ABB RobotStudio station: TEST1_20190225-105659.rsstn

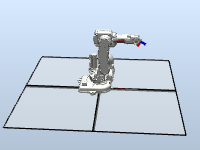
Station TEST1 (saved by RobotStudio 6.8.8148.134)
Controller IRB_140_6kg_0.81m
  mechanical unit ROB_1: IRB140_6_81_C_03, 6 joints, base frame (0, 0, 0) mm
Layout (positions relative to the parent item):
  - IRB140_6_81_C_03 [mechanism, from Robots\IRB140_6_81_C_G_03.rslib] at (0, 0, 0) mm; joint values [0, 0, 0, 0, 0.5236, 0] (rad or m)
